// TIA Portal V17 export
// export: Created 2025-05-22T06:01:52.5137085Z, ExportSetting WithDefaults, DisplayName Totally Integrated Automation Portal, DisplayVersion V17 Update 8, DisplayName TIA Portal Openness, DisplayVersion V17 Update 8, DisplayName TIA Portal Version Control Interface, DisplayVersion V17, DisplayName SINAMICS Startdrive Advanced, DisplayVersion V17 SP2, DisplayName SINAMICS Startdrive G110M, G120, G120C, G120D, G120P, G115D, DisplayVersion V17 SP2, DisplayName SINAMICS Startdrive G130, G150, S120, S150, SINAMICS MV, S210, DisplayVersion V17 SP2, DisplayName STEP 7 Professional, DisplayVersion V17 Update 8, DisplayName SINUMERIK ONE STEP 7 Toolbox, DisplayVersion V17 Update 12, DisplayName SINUMERIK ONE PLC Basic Program Plus, DisplayVersion V17 Update 12, DisplayName SINUMERIK 840D sl STEP 7 Toolbox, DisplayVersion V17 Update 12, DisplayName STEP 7 Safety, DisplayVersion V17 Update 6, DisplayName WinCC Advanced, DisplayVersion V17 Update 8
FUNCTION "UPTL_EnergyConsumption" : Void   // FC1058, LAD
TITLE = UPTL_EnergyConsumption / UPTL_EnergyCosumption
{ S7_Optimized_Access := 'FALSE' }
AUTHOR : Transline
FAMILY : UPTL_Transline
VERSION : 17.0
// Beispiel für den Aufruf der Funktionen aus HMIEnergyData
// stored: AutoNumber true, IsIECCheckEnabled false, SetENOAutomatically false, UDAEnableTagReadback false
BEGIN

REGION Network 1
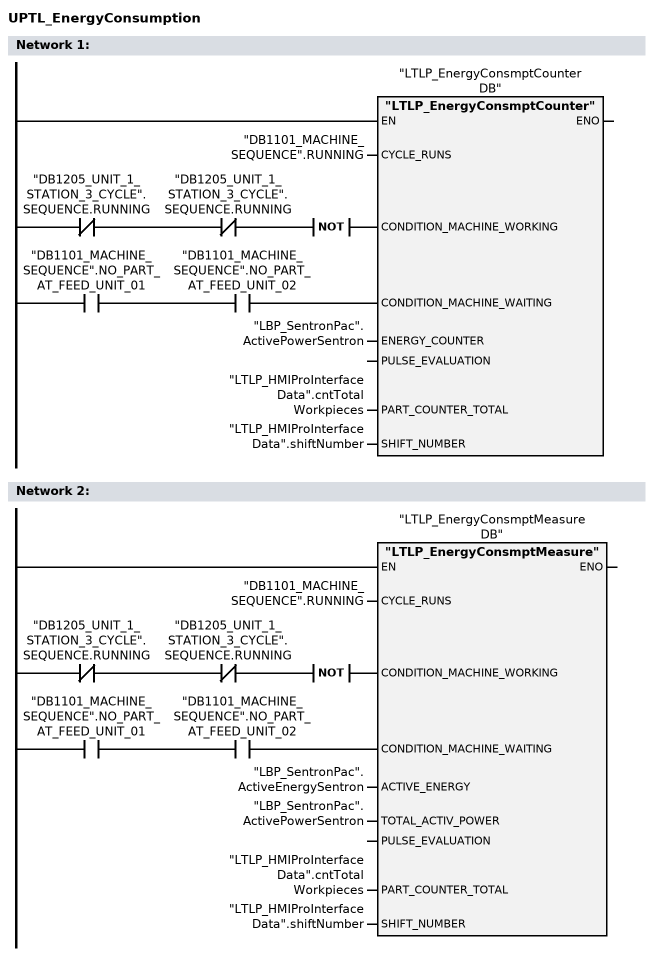
   RUNG wire#powerrail
      "LTLP_EnergyConsmptCounterDB"(CONDITION_MACHINE_WORKING := wire#w1, CONDITION_MACHINE_WAITING := wire#w2, CYCLE_RUNS := "DB1101_MACHINE_SEQUENCE".RUNNING, ENERGY_COUNTER := "LBP_SentronPac".ActivePowerSentron, PULSE_EVALUATION :=, PART_COUNTER_TOTAL := "LTLP_HMIProInterfaceData".cntTotalWorkpieces, SHIFT_NUMBER := "LTLP_HMIProInterfaceData".shiftNumber)
   END_RUNG
   RUNG wire#powerrail
      I_Contact( "DB1205_UNIT_1_STATION_3_CYCLE".SEQUENCE.RUNNING )
      I_Contact( "DB1205_UNIT_1_STATION_3_CYCLE".SEQUENCE.RUNNING )
      Not()
   END_RUNG wire#w1
   RUNG wire#powerrail
      Contact( "DB1101_MACHINE_SEQUENCE".NO_PART_AT_FEED_UNIT_01 )
      Contact( "DB1101_MACHINE_SEQUENCE".NO_PART_AT_FEED_UNIT_02 )
   END_RUNG wire#w2
   // the same network as SCL:
   "LTLP_EnergyConsmptCounterDB"(CYCLE_RUNS := "DB1101_MACHINE_SEQUENCE".RUNNING,   // "LTLP_EnergyConsmptCounter"
                           CONDITION_MACHINE_WORKING := NOT (NOT "DB1205_UNIT_1_STATION_3_CYCLE".SEQUENCE.RUNNING AND NOT "DB1205_UNIT_1_STATION_3_CYCLE".SEQUENCE.RUNNING),
                           CONDITION_MACHINE_WAITING := "DB1101_MACHINE_SEQUENCE".NO_PART_AT_FEED_UNIT_01 AND "DB1101_MACHINE_SEQUENCE".NO_PART_AT_FEED_UNIT_02,
                           ENERGY_COUNTER := "LBP_SentronPac".ActivePowerSentron,
                           PART_COUNTER_TOTAL := "LTLP_HMIProInterfaceData".cntTotalWorkpieces,
                           SHIFT_NUMBER := "LTLP_HMIProInterfaceData".shiftNumber);
END_REGION

REGION Network 2
   RUNG wire#powerrail
      "LTLP_EnergyConsmptMeasureDB"(CONDITION_MACHINE_WORKING := wire#w1, CONDITION_MACHINE_WAITING := wire#w2, CYCLE_RUNS := "DB1101_MACHINE_SEQUENCE".RUNNING, ACTIVE_ENERGY := "LBP_SentronPac".ActiveEnergySentron, TOTAL_ACTIV_POWER := "LBP_SentronPac".ActivePowerSentron, PULSE_EVALUATION :=, PART_COUNTER_TOTAL := "LTLP_HMIProInterfaceData".cntTotalWorkpieces, SHIFT_NUMBER := "LTLP_HMIProInterfaceData".shiftNumber)
   END_RUNG
   RUNG wire#powerrail
      I_Contact( "DB1205_UNIT_1_STATION_3_CYCLE".SEQUENCE.RUNNING )
      I_Contact( "DB1205_UNIT_1_STATION_3_CYCLE".SEQUENCE.RUNNING )
      Not()
   END_RUNG wire#w1
   RUNG wire#powerrail
      Contact( "DB1101_MACHINE_SEQUENCE".NO_PART_AT_FEED_UNIT_01 )
      Contact( "DB1101_MACHINE_SEQUENCE".NO_PART_AT_FEED_UNIT_02 )
   END_RUNG wire#w2
   // the same network as SCL:
   "LTLP_EnergyConsmptMeasureDB"(CYCLE_RUNS := "DB1101_MACHINE_SEQUENCE".RUNNING,   // "LTLP_EnergyConsmptMeasure"
                           CONDITION_MACHINE_WORKING := NOT (NOT "DB1205_UNIT_1_STATION_3_CYCLE".SEQUENCE.RUNNING AND NOT "DB1205_UNIT_1_STATION_3_CYCLE".SEQUENCE.RUNNING),
                           CONDITION_MACHINE_WAITING := "DB1101_MACHINE_SEQUENCE".NO_PART_AT_FEED_UNIT_01 AND "DB1101_MACHINE_SEQUENCE".NO_PART_AT_FEED_UNIT_02,
                           ACTIVE_ENERGY := "LBP_SentronPac".ActiveEnergySentron,
                           TOTAL_ACTIV_POWER := "LBP_SentronPac".ActivePowerSentron,
                           PART_COUNTER_TOTAL := "LTLP_HMIProInterfaceData".cntTotalWorkpieces,
                           SHIFT_NUMBER := "LTLP_HMIProInterfaceData".shiftNumber);
END_REGION
END_FUNCTION
